FUNCTION_BLOCK FB_Glowny
VAR
	iRuchX:INT:=50;
	iRuchY:INT:=50;
	predkoscRuchu:TIME:=T#2MS;
	czasoOdmierzacz:TON;
	timerRuchu:TON;
	iStan: INT;
END_VAR

CASE iStan OF
	
0:
	czasoOdmierzacz(IN:=TRUE, PT:=(predkoscRuchu/100));
	IF czasoOdmierzacz.Q=TRUE THEN
		iRuchY:=iRuchY+1;
		czasoOdmierzacz(IN:=FALSE);
	END_IF
	IF iRuchY=600 THEN
		iStan:=1;
	END_IF

1:
	czasoOdmierzacz(IN:=TRUE, PT:=(predkoscRuchu/100));
	IF czasoOdmierzacz.Q=TRUE THEN
		iRuchX:=iRuchX+1;
		czasoOdmierzacz(IN:=FALSE);
	END_IF
	IF iRuchX=1100 THEN
		iStan:=2;
	END_IF

2:
	czasoOdmierzacz(IN:=TRUE, PT:=(predkoscRuchu/100));
	IF czasoOdmierzacz.Q=TRUE THEN
		iRuchY:=iRuchY-1;
		czasoOdmierzacz(IN:=FALSE);
	END_IF
	IF iRuchY=50 THEN
		iStan:=3;
	END_IF


3:
	czasoOdmierzacz(IN:=TRUE, PT:=(predkoscRuchu/100));
	IF czasoOdmierzacz.Q=TRUE THEN
		iRuchX:=iRuchX-1;
		czasoOdmierzacz(IN:=FALSE);
	END_IF
	IF iRuchX=50 THEN
		iStan:=0;
	END_IF


END_CASE

END_FUNCTION_BLOCK

(* stored: Version 1.1.0.1, ProductVersion 3.1.4024.4
   POU FB_Glowny: Id {12d3453c-e68a-4d1f-ae44-22ee6a2954e9}, SpecialFunc None *)
